  MoveL 1958 to (-198.35, 431.99, -17.53) mm, rotated rx 180 ry 0 rz 13.34 deg; joints [-4.464, -30.989, 133.935, -182.853, 90.229, 89.268, 155.338]
  MoveL 1959 to (-199.1, 431.99, -17.53) mm, rotated rx -180 ry 0 rz 13.42 deg; joints [-4.464, -30.964, 133.923, -182.853, 90.243, 89.268, 155.256]
  MoveL 1960 to (-199.28, 431.98, -17.52) mm, rotated rx 180 ry 0 rz 13.44 deg; joints [-4.464, -30.958, 133.921, -182.853, 90.246, 89.267, 155.235]
  MoveL 1961 to (-199.47, 431.96, -17.53) mm, rotated rx -180 ry 0 rz 13.47 deg; joints [-4.464, -30.953, 133.919, -182.853, 90.249, 89.267, 155.213]
  MoveL 1962 to (-199.66, 431.92, -17.53) mm, rotated rx -180 ry 0 rz 13.49 deg; joints [-4.464, -30.95, 133.917, -182.853, 90.251, 89.267, 155.191]
  MoveL 1963 to (-199.85, 431.88, -17.52) mm, rotated rx -180 ry 0 rz 13.51 deg; joints [-4.464, -30.947, 133.916, -182.853, 90.252, 89.267, 155.168]
  MoveL 1964 to (-200.27, 431.74, -17.52) mm, rotated rx 180 ry 0 rz 13.57 deg; joints [-4.464, -30.942, 133.913, -182.853, 90.255, 89.267, 155.115]
  MoveL 1965 to (-204.13, 430.52, -17.53) mm, rotated rx 180 ry 0 rz 14.05 deg; joints [-4.464, -30.898, 133.894, -182.854, 90.279, 89.266, 154.632]
  MoveL 1966 to (-204.42, 430.43, -17.53) mm, rotated rx 180 ry 0 rz 14.08 deg; joints [-4.464, -30.895, 133.892, -182.854, 90.28, 89.266, 154.595]
  MoveL 1967 to (-204.57, 430.37, -17.52) mm, rotated rx 180 ry 0 rz 14.1 deg; joints [-4.464, -30.894, 133.892, -182.854, 90.281, 89.266, 154.577]
  MoveL 1968 to (-204.72, 430.31, -17.53) mm, rotated rx 180 ry 0 rz 14.12 deg; joints [-4.464, -30.894, 133.892, -182.854, 90.281, 89.266, 154.557]
  MoveL 1969 to (-204.86, 430.23, -17.53) mm, rotated rx -180 ry 0 rz 14.14 deg; joints [-4.464, -30.894, 133.892, -182.854, 90.281, 89.266, 154.538]
  MoveL 1970 to (-205.01, 430.15, -17.53) mm, rotated rx 180 ry 0 rz 14.16 deg; joints [-4.464, -30.896, 133.892, -182.854, 90.28, 89.266, 154.517]
  MoveL 1971 to (-205.16, 430.05, -17.53) mm, rotated rx 180 ry 0 rz 14.18 deg; joints [-4.464, -30.897, 133.893, -182.854, 90.279, 89.266, 154.497]
  MoveL 1972 to (-205.3, 429.94, -17.52) mm, rotated rx 180 ry 0 rz 14.2 deg; joints [-4.464, -30.9, 133.895, -182.854, 90.278, 89.266, 154.475]
  MoveL 1973 to (-205.53, 429.75, -17.52) mm, rotated rx 180 ry 0 rz 14.24 deg; joints [-4.464, -30.906, 133.897, -182.854, 90.274, 89.266, 154.441]
  MoveL 1974 to (-205.75, 429.52, -17.52) mm, rotated rx 180 ry 0 rz 14.28 deg; joints [-4.464, -30.916, 133.902, -182.854, 90.269, 89.266, 154.404]
  MoveL 1975 to (-205.92, 429.3, -17.52) mm, rotated rx -180 ry 0 rz 14.3 deg; joints [-4.464, -30.925, 133.906, -182.854, 90.264, 89.267, 154.375]
  MoveL 1976 to (-206.06, 429.09, -17.53) mm, rotated rx -180 ry 0 rz 14.33 deg; joints [-4.464, -30.936, 133.911, -182.853, 90.258, 89.267, 154.348]
  MoveL 1977 to (-206.14, 428.95, -17.53) mm, rotated rx -180 ry 0 rz 14.35 deg; joints [-4.464, -30.943, 133.914, -182.853, 90.254, 89.267, 154.333]
  MoveL 1978 to (-206.21, 428.82, -17.52) mm, rotated rx 180 ry 0 rz 14.36 deg; joints [-4.464, -30.951, 133.917, -182.853, 90.25, 89.267, 154.319]
  MoveL 1979 to (-206.27, 428.69, -17.53) mm, rotated rx 180 ry 0 rz 14.37 deg; joints [-4.464, -30.958, 133.921, -182.853, 90.246, 89.267, 154.305]
  MoveL 1980 to (-206.32, 428.55, -17.53) mm, rotated rx 180 ry 0 rz 14.39 deg; joints [-4.464, -30.966, 133.925, -182.853, 90.242, 89.268, 154.292]
  MoveL 1981 to (-206.37, 428.42, -17.53) mm, rotated rx 180 ry 0 rz 14.4 deg; joints [-4.464, -30.975, 133.928, -182.853, 90.237, 89.268, 154.28]
  MoveL 1982 to (-206.41, 428.28, -17.52) mm, rotated rx -180 ry 0 rz 14.41 deg; joints [-4.464, -30.983, 133.932, -182.853, 90.233, 89.268, 154.268]
  MoveL 1983 to (-206.47, 428.01, -17.53) mm, rotated rx -180 ry 0 rz 14.43 deg; joints [-4.464, -31.001, 133.94, -182.853, 90.223, 89.269, 154.248]
  MoveL 1984 to (-206.5, 427.77, -17.53) mm, rotated rx 180 ry 0 rz 14.45 deg; joints [-4.464, -31.017, 133.948, -182.853, 90.214, 89.269, 154.231]
  MoveL 1985 to (-206.52, 427.53, -17.53) mm, rotated rx 180 ry 0 rz 14.46 deg; joints [-4.464, -31.034, 133.955, -182.853, 90.205, 89.27, 154.217]
  MoveL 1986 to (-206.52, 427.04, -17.53) mm, rotated rx 180 ry 0 rz 14.49 deg; joints [-4.464, -31.069, 133.971, -182.853, 90.185, 89.27, 154.191]
  MoveL 1987 to (-206.52, 50.21, -17.53) mm, rotated rx 180 ry 0 rz 65.02 deg; joints [-4.427, -53.233, 140.509, -182.923, 74.579, 90.066, 103.664]
  MoveL 1988 to (-206.51, 49.73, -17.52) mm, rotated rx 180 ry 0 rz 65.14 deg; joints [-4.427, -53.244, 140.51, -182.923, 74.569, 90.066, 103.539]
  MoveL 1989 to (-206.48, 49.48, -17.53) mm, rotated rx 180 ry 0 rz 65.2 deg; joints [-4.427, -53.252, 140.511, -182.923, 74.563, 90.066, 103.477]
  MoveL 1990 to (-206.43, 49.24, -17.53) mm, rotated rx -180 ry 0 rz 65.26 deg; joints [-4.427, -53.26, 140.513, -182.923, 74.555, 90.067, 103.417]
  MoveL 1991 to (-206.37, 49.02, -17.53) mm, rotated rx -180 ry 0 rz 65.32 deg; joints [-4.427, -53.27, 140.514, -182.923, 74.547, 90.067, 103.362]
  MoveL 1992 to (-206.28, 48.8, -17.53) mm, rotated rx -180 ry 0 rz 65.37 deg; joints [-4.427, -53.281, 140.516, -182.923, 74.537, 90.068, 103.309]
  MoveL 1993 to (-206.18, 48.57, -17.53) mm, rotated rx 180 ry 0 rz 65.42 deg; joints [-4.427, -53.294, 140.517, -182.924, 74.526, 90.068, 103.256]
  MoveL 1994 to (-206.06, 48.35, -17.52) mm, rotated rx 180 ry 0 rz 65.47 deg; joints [-4.427, -53.309, 140.519, -182.924, 74.514, 90.069, 103.205]
  MoveL 1995 to (-205.98, 48.22, -17.52) mm, rotated rx 180 ry 0 rz 65.5 deg; joints [-4.427, -53.319, 140.521, -182.924, 74.505, 90.07, 103.176]
  MoveL 1996 to (-205.88, 48.09, -17.52) mm, rotated rx 180 ry 0 rz 65.53 deg; joints [-4.427, -53.329, 140.522, -182.924, 74.497, 90.07, 103.148]
  MoveL 1997 to (-205.78, 47.96, -17.53) mm, rotated rx -180 ry 0 rz 65.56 deg; joints [-4.427, -53.34, 140.524, -182.924, 74.487, 90.071, 103.12]
  MoveL 1998 to (-205.66, 47.83, -17.52) mm, rotated rx 180 ry 0 rz 65.59 deg; joints [-4.427, -53.352, 140.525, -182.924, 74.477, 90.071, 103.092]
  MoveL 1999 to (-205.51, 47.67, -17.52) mm, rotated rx 180 ry 0 rz 65.62 deg; joints [-4.427, -53.369, 140.528, -182.924, 74.463, 90.072, 103.06]
  MoveL 2000 to (-205.35, 47.54, -17.53) mm, rotated rx -180 ry 0 rz 65.65 deg; joints [-4.427, -53.384, 140.53, -182.924, 74.449, 90.073, 103.034]
  MoveL 2001 to (-205.19, 47.42, -17.52) mm, rotated rx 180 ry 0 rz 65.67 deg; joints [-4.427, -53.4, 140.532, -182.925, 74.436, 90.073, 103.012]
  MoveL 2002 to (-205.03, 47.31, -17.52) mm, rotated rx 180 ry 0 rz 65.69 deg; joints [-4.427, -53.415, 140.534, -182.925, 74.422, 90.074, 102.993]
  MoveL 2003 to (-204.81, 47.18, -17.53) mm, rotated rx -180 ry 0 rz 65.71 deg; joints [-4.427, -53.437, 140.537, -182.925, 74.404, 90.075, 102.973]
  MoveL 2004 to (-204.58, 47.08, -17.53) mm, rotated rx -180 ry 0 rz 65.72 deg; joints [-4.427, -53.458, 140.54, -182.925, 74.386, 90.076, 102.958]
  MoveL 2005 to (-204.36, 46.99, -17.52) mm, rotated rx 180 ry 0 rz 65.73 deg; joints [-4.427, -53.478, 140.543, -182.925, 74.368, 90.077, 102.95]
  MoveL 2006 to (-204.13, 46.92, -17.53) mm, rotated rx -180 ry 0 rz 65.73 deg; joints [-4.427, -53.498, 140.546, -182.926, 74.351, 90.078, 102.946]
  MoveL 2007 to (-203.89, 46.87, -17.53) mm, rotated rx -180 ry 0 rz 65.73 deg; joints [-4.427, -53.519, 140.549, -182.926, 74.333, 90.079, 102.947]
  MoveL 2008 to (-203.65, 46.84, -17.53) mm, rotated rx -180 ry 0 rz 65.73 deg; joints [-4.427, -53.54, 140.552, -182.926, 74.315, 90.08, 102.953]
  MoveL 2009 to (-203.41, 46.83, -17.52) mm, rotated rx 180 ry 0 rz 65.72 deg; joints [-4.427, -53.561, 140.554, -182.926, 74.297, 90.081, 102.964]
  MoveL 2010 to (-203.17, 46.82, -17.53) mm, rotated rx -180 ry 0 rz 65.7 deg; joints [-4.427, -53.581, 140.557, -182.927, 74.28, 90.081, 102.979]
  MoveL 2011 to (222.09, 46.83, -17.53) mm, rotated rx 180 ry 0 rz -49.41 deg; joints [-4.71, -87.722, 145.676, -197.389, 6.41, 104.735, 179]
  MoveL 2012 to (223.29, 46.83, -17.53) mm, rotated rx -180 ry 0 rz -49.48 deg; joints [-4.713, -87.801, 145.732, -197.613, 6.328, 104.955, 179]
  MoveL 2013 to (223.53, 46.84, -17.53) mm, rotated rx -180 ry 0 rz -49.49 deg; joints [-4.713, -87.816, 145.745, -197.643, 6.318, 104.985, 179]
  MoveL 2014 to (223.77, 46.87, -17.53) mm, rotated rx 180 ry 0 rz -49.49 deg; joints [-4.714, -87.83, 145.76, -197.653, 6.315, 104.995, 179]
  MoveL 2015 to (224.01, 46.92, -17.53) mm, rotated rx 180 ry 0 rz -49.49 deg; joints [-4.715, -87.843, 145.778, -197.643, 6.32, 104.984, 179]
  MoveL 2016 to (224.24, 46.99, -17.53) mm, rotated rx 180 ry 0 rz -49.49 deg; joints [-4.716, -87.853, 145.797, -197.615, 6.333, 104.954, 179]
  MoveL 2017 to (224.46, 47.08, -17.53) mm, rotated rx -180 ry 0 rz -49.48 deg; joints [-4.717, -87.863, 145.819, -197.566, 6.353, 104.905, 179]
  MoveL 2018 to (224.69, 47.18, -17.53) mm, rotated rx -180 ry 0 rz -49.46 deg; joints [-4.718, -87.872, 145.843, -197.496, 6.382, 104.834, 179]
  MoveL 2019 to (224.92, 47.31, -17.53) mm, rotated rx -180 ry 0 rz -49.44 deg; joints [-4.719, -87.879, 145.87, -197.403, 6.42, 104.74, 179]
  MoveL 2020 to (225.07, 47.42, -17.53) mm, rotated rx 180 ry 0 rz -49.42 deg; joints [-4.72, -87.883, 145.891, -197.323, 6.454, 104.659, 179]
  MoveL 2021 to (225.23, 47.54, -17.53) mm, rotated rx 180 ry 0 rz -49.4 deg; joints [-4.721, -87.886, 145.913, -197.229, 6.493, 104.564, 179]
  MoveL 2022 to (225.39, 47.67, -17.53) mm, rotated rx -180 ry 0 rz -49.38 deg; joints [-4.722, -87.888, 145.938, -197.119, 6.54, 104.454, 179]
  MoveL 2023 to (225.55, 47.83, -17.53) mm, rotated rx 180 ry 0 rz -49.35 deg; joints [-4.723, -87.889, 145.966, -196.991, 6.595, 104.325, 179]
  MoveL 2024 to (225.66, 47.96, -17.52) mm, rotated rx -180 ry 0 rz -49.32 deg; joints [-4.724, -87.888, 145.988, -196.884, 6.641, 104.217, 179]
  MoveL 2025 to (225.77, 48.09, -17.52) mm, rotated rx 180 ry 0 rz -49.3 deg; joints [-4.724, -87.887, 146.009, -196.777, 6.688, 104.109, 179]
  MoveL 2026 to (225.86, 48.22, -17.52) mm, rotated rx 180 ry 0 rz -49.27 deg; joints [-4.725, -87.885, 146.03, -196.669, 6.736, 104.001, 179]
  MoveL 2027 to (225.94, 48.35, -17.53) mm, rotated rx -180 ry 0 rz -49.24 deg; joints [-4.726, -87.883, 146.051, -196.562, 6.785, 103.893, 179]
  MoveL 2028 to (226.07, 48.57, -17.53) mm, rotated rx -180 ry 0 rz -49.19 deg; joints [-4.727, -87.877, 146.085, -196.378, 6.869, 103.709, 179]
  MoveL 2029 to (226.17, 48.8, -17.53) mm, rotated rx -180 ry 0 rz -49.15 deg; joints [-4.728, -87.87, 146.118, -196.196, 6.955, 103.525, 179]
  MoveL 2030 to (226.25, 49.02, -17.53) mm, rotated rx 180 ry 0 rz -49.1 deg; joints [-4.729, -87.861, 146.15, -196.015, 7.043, 103.343, 179]
  MoveL 2031 to (226.31, 49.24, -17.53) mm, rotated rx 180 ry 0 rz -49.04 deg; joints [-4.73, -87.852, 146.181, -195.836, 7.132, 103.163, 179]
  MoveL 2032 to (226.36, 49.48, -17.52) mm, rotated rx -180 ry 0 rz -48.99 deg; joints [-4.731, -87.84, 146.214, -195.643, 7.229, 102.97, 179]
  MoveL 2033 to (226.39, 49.73, -17.53) mm, rotated rx -180 ry 0 rz -48.93 deg; joints [-4.733, -87.826, 146.246, -195.453, 7.329, 102.78, 179]
  MoveL 2034 to (226.4, 50.21, -17.52) mm, rotated rx 180 ry 0 rz -48.82 deg; joints [-4.735, -87.796, 146.308, -195.082, 7.531, 102.406, 179]
  MoveL 2035 to (226.4, 428.01, -17.53) mm, rotated rx -180 ry 0 rz -39.2 deg; joints [-4.974, -49.079, 151.02, -182.914, 60.345, 89.094, 179]
  MoveL 2036 to (226.4, 428.98, -17.53) mm, rotated rx 180 ry 0 rz -39.14 deg; joints [-4.975, -48.95, 151.007, -182.912, 60.515, 89.088, 179]
  MoveL 2037 to (226.38, 429.22, -17.52) mm, rotated rx 180 ry 0 rz -39.13 deg; joints [-4.975, -48.917, 151.002, -182.912, 60.559, 89.086, 179]
  MoveL 2038 to (226.34, 429.46, -17.53) mm, rotated rx -180 ry 0 rz -39.11 deg; joints [-4.975, -48.882, 150.997, -182.911, 60.606, 89.085, 179]
  MoveL 2039 to (226.28, 429.7, -17.53) mm, rotated rx -180 ry 0 rz -39.09 deg; joints [-4.975, -48.847, 150.991, -182.911, 60.654, 89.083, 179]
  MoveL 2040 to (226.2, 429.94, -17.53) mm, rotated rx 180 ry 0 rz -39.07 deg; joints [-4.975, -48.811, 150.983, -182.911, 60.704, 89.082, 179]
  MoveL 2041 to (226.15, 430.07, -17.53) mm, rotated rx -180 ry 0 rz -39.06 deg; joints [-4.975, -48.791, 150.978, -182.91, 60.733, 89.081, 179]
  MoveL 2042 to (226.09, 430.21, -17.53) mm, rotated rx -180 ry 0 rz -39.04 deg; joints [-4.975, -48.77, 150.973, -182.91, 60.762, 89.08, 179]
  MoveL 2043 to (226.02, 430.34, -17.53) mm, rotated rx -180 ry 0 rz -39.03 deg; joints [-4.975, -48.749, 150.968, -182.91, 60.791, 89.079, 179]
  MoveL 2044 to (225.94, 430.47, -17.53) mm, rotated rx 180 ry 0 rz -39.01 deg; joints [-4.975, -48.728, 150.962, -182.91, 60.822, 89.079, 179]
  MoveL 2045 to (225.78, 430.71, -17.53) mm, rotated rx 180 ry 0 rz -38.98 deg; joints [-4.975, -48.687, 150.95, -182.91, 60.881, 89.077, 179]
  MoveL 2046 to (225.58, 430.96, -17.52) mm, rotated rx 180 ry 0 rz -38.95 deg; joints [-4.975, -48.645, 150.936, -182.909, 60.944, 89.076, 179]
  MoveL 2047 to (225.44, 431.1, -17.53) mm, rotated rx 180 ry 0 rz -38.93 deg; joints [-4.975, -48.618, 150.927, -182.909, 60.983, 89.075, 179]
  MoveL 2048 to (225.3, 431.23, -17.53) mm, rotated rx -180 ry 0 rz -38.91 deg; joints [-4.975, -48.594, 150.917, -182.909, 61.02, 89.075, 179]
  MoveL 2049 to (225.16, 431.34, -17.52) mm, rotated rx 180 ry 0 rz -38.88 deg; joints [-4.974, -48.572, 150.908, -182.909, 61.054, 89.074, 179]
  MoveL 2050 to (225.02, 431.44, -17.52) mm, rotated rx -180 ry 0 rz -38.86 deg; joints [-4.974, -48.551, 150.899, -182.909, 61.085, 89.074, 179]
  MoveL 2051 to (224.78, 431.59, -17.53) mm, rotated rx -180 ry 0 rz -38.83 deg; joints [-4.974, -48.521, 150.885, -182.908, 61.134, 89.073, 179]
  MoveL 2052 to (224.55, 431.71, -17.52) mm, rotated rx 180 ry 0 rz -38.8 deg; joints [-4.973, -48.493, 150.871, -182.908, 61.178, 89.073, 179]
  MoveL 2053 to (224.32, 431.8, -17.53) mm, rotated rx -180 ry 0 rz -38.77 deg; joints [-4.973, -48.469, 150.857, -182.908, 61.218, 89.072, 179]
  MoveL 2054 to (224.09, 431.88, -17.53) mm, rotated rx -180 ry 0 rz -38.74 deg; joints [-4.973, -48.447, 150.844, -182.908, 61.254, 89.072, 179]
  MoveL 2055 to (224.01, 431.9, -17.53) mm, rotated rx -180 ry 0 rz -38.74 deg; joints [-4.972, -48.441, 150.84, -182.908, 61.265, 89.072, 179]
  MoveL 2056 to (223.77, 431.95, -17.53) mm, rotated rx -180 ry 0 rz -38.71 deg; joints [-4.972, -48.422, 150.826, -182.908, 61.299, 89.072, 179]
  MoveL 2057 to (223.53, 431.98, -17.53) mm, rotated rx 180 ry 0 rz -38.68 deg; joints [-4.971, -48.405, 150.813, -182.908, 61.329, 89.073, 179]
  MoveL 2058 to (223.29, 431.99, -17.53) mm, rotated rx -180 ry 0 rz -38.65 deg; joints [-4.971, -48.391, 150.8, -182.908, 61.356, 89.073, 179]
  MoveL 2059 to (223.05, 431.99, -17.53) mm, rotated rx 180 ry 0 rz -38.63 deg; joints [-4.97, -48.379, 150.787, -182.908, 61.38, 89.073, 179]
  MoveL 2060 to (-164.9, 431.99, -17.52) mm, rotated rx 180 ry 0 rz 9.57 deg; joints [-4.462, -32.044, 134.405, -182.852, 89.645, 89.298, 159.107]
  MoveL 2061 to (-194.97, 431.99, -17.52) mm, rotated rx 180 ry 0 rz 12.97 deg; joints [-4.464, -31.102, 133.986, -182.853, 90.167, 89.271, 155.709]
  MoveL 2062 to (-195.47, 431.99, -17.52) mm, rotated rx 180 ry 0 rz 13.03 deg; joints [-4.464, -31.086, 133.979, -182.853, 90.176, 89.271, 155.654]
  Set speed (38.1 mm/s)
  MoveL 2063 to (-196.09, 432.77, -17.52) mm, rotated rx -180 ry 0 rz 13.06 deg; joints [-4.464, -31.008, 133.943, -182.853, 90.219, 89.269, 155.625]
  MoveL 2064 to (-195.65, 434.72, -17.53) mm, rotated rx 180 ry 0 rz 12.91 deg; joints [-4.464, -30.878, 133.885, -182.854, 90.29, 89.265, 155.769]
  MoveL 2065 to (-195.51, 435.34, -16.89) mm, rotated rx 180 ry 0 rz 12.86 deg; joints [-4.429, -30.837, 133.868, -182.819, 90.315, 89.272, 155.815]
  Set speed (100.0 mm/s)
  MoveL 2066 to (-195.51, 435.34, 34.52) mm, rotated rx 180 ry 0 rz 12.86 deg; joints [-1.585, -30.826, 133.954, -180.045, 90.428, 89.913, 155.815]
  MoveL 2067 to (-195.51, 435.34, 34.52) mm, rotated rx 180 ry 0 rz 12.86 deg; joints [-1.585, -30.826, 133.954, -180.045, 90.428, 89.913, 155.815]
